(* Logix 5000 project; controller TEC_81 vendor 1 type 14 code 148 rev 36.11; software revision 36.00; part 4 of 4 *)
(* tags used below, declared in another part *)
   Safety_Close_Loop_ok : BOOL;
   TOF_STO_KinetixStorage1 : TIMER;
   Abrir_Prensa_CNC_1_Safety : BOOL;   // Abrir Prensa CNC 1
   Abrir_Prensa_CNC_2_Safety : BOOL;
   Cerrar_Prensa_CNC_1_Safety : BOOL;   // Cerrar Prensa CNC 1
   Cerrar_Prensa_CNC_2_Safety : BOOL;
   Close_Door_CNC_1_Safety : BOOL;   // Cerrar Puerta de CNC 1 Desde ArmorBlock
   Close_Door_CNC_2_Safety : BOOL;   // Cerrar Puerta de CNC 2 Desde ArmorBlock
   CycleStartDly : TIMER;
   EStops_OK : BOOL;
   Interlocks_Ok : BOOL;
   KUKA : TIMER;
   LigthCurtain_ok : BOOL;
   Paro_Emergencia_Almacen_1 : BOOL;   // Señal de paro para Torc Off Almacen 1
   Paro_Emergencia_Almacen_2 : BOOL;   // Señal de paro para Torc Off Almacen 2
   Pulse : TIMER;
   Reset_Almacen_1_Sfty : BOOL;
   Reset_Almacen_2_Sfty : BOOL;
   Reset_Principal_Sfty : BOOL;
   Reset_Salida_1_Sfty : BOOL;
   Safety_Test_Bit : DINT;
   SafetyReset_almacen_1 : BOOL;
   SafetyReset_almacen_2 : BOOL;
   SafetyReset_Principal : BOOL;
   SafetyReset_Salida_1 : BOOL;
   Storage_2 : BOOL;
   Storage_3 : BOOL;
   Storage_4 : BOOL;
   Storage_5 : BOOL;
   TOF_STO_KinetixStorage2 : TIMER;
   TT : BOOL;
(* SafetyProgram, continued *)

ROUTINE MainRoutine   (* ladder *)
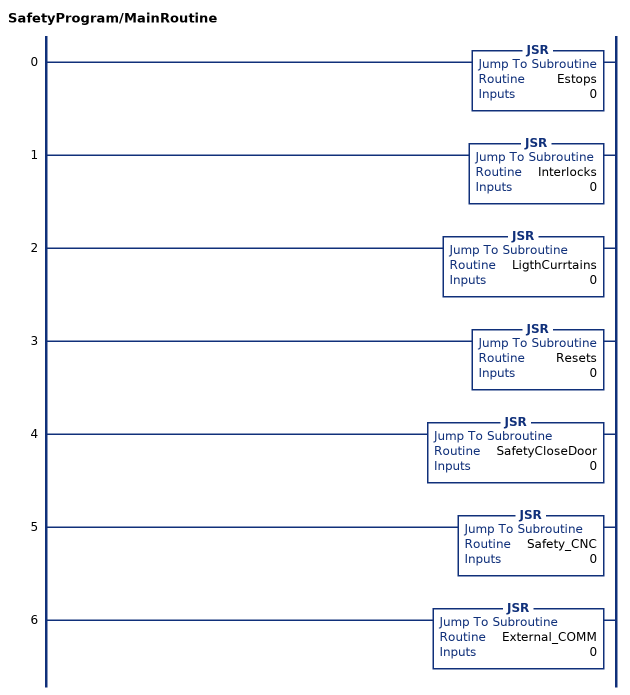
   0: JSR(Estops,0);
   1: JSR(Interlocks,0);
   2: JSR(LigthCurrtains,0);
   3: JSR(Resets,0);
   4: JSR(SafetyCloseDoor,0);
   5: JSR(Safety_CNC,0);
   6: JSR(External_COMM,0);
END_ROUTINE

ROUTINE Resets   (* ladder *)
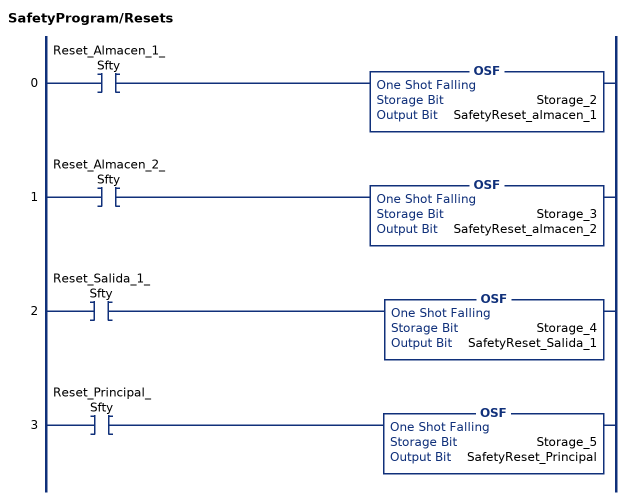
   0: XIC(Reset_Almacen_1_Sfty)OSF(Storage_2,SafetyReset_almacen_1);
   1: XIC(Reset_Almacen_2_Sfty)OSF(Storage_3,SafetyReset_almacen_2);
   2: XIC(Reset_Salida_1_Sfty)OSF(Storage_4,SafetyReset_Salida_1);
   3: XIC(Reset_Principal_Sfty)OSF(Storage_5,SafetyReset_Principal);
END_ROUTINE

ROUTINE Safety_CNC   (* ladder *)
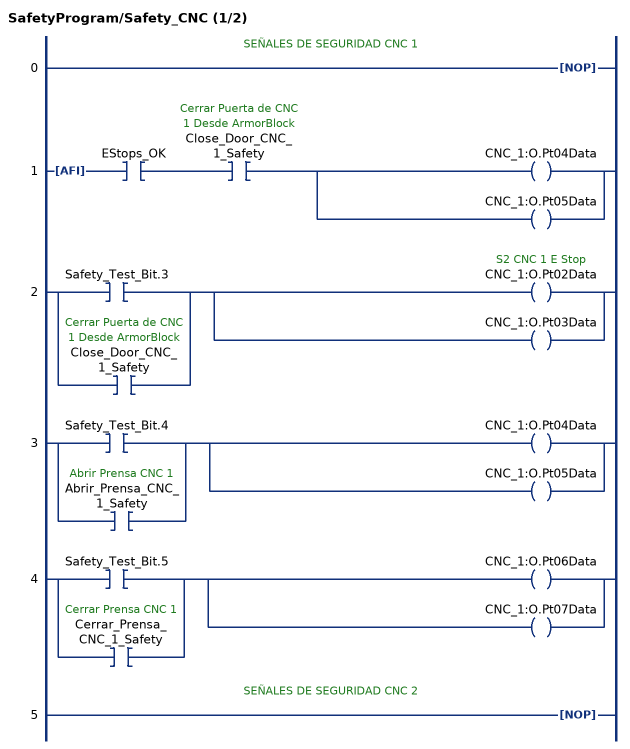
   // SEÑALES DE SEGURIDAD CNC 1
   0: NOP();
   1: AFI()XIC(EStops_OK)XIC(Close_Door_CNC_1_Safety)[OTE(CNC_1:O.Pt04Data) ,OTE(CNC_1:O.Pt05Data) ];
   2: [XIC(Safety_Test_Bit.3) ,XIC(Close_Door_CNC_1_Safety) ][OTE(CNC_1:O.Pt02Data) ,OTE(CNC_1:O.Pt03Data) ];
   3: [XIC(Safety_Test_Bit.4) ,XIC(Abrir_Prensa_CNC_1_Safety) ][OTE(CNC_1:O.Pt04Data) ,OTE(CNC_1:O.Pt05Data) ];
   4: [XIC(Safety_Test_Bit.5) ,XIC(Cerrar_Prensa_CNC_1_Safety) ][OTE(CNC_1:O.Pt06Data) ,OTE(CNC_1:O.Pt07Data) ];
   // SEÑALES DE SEGURIDAD CNC 2
   5: NOP();
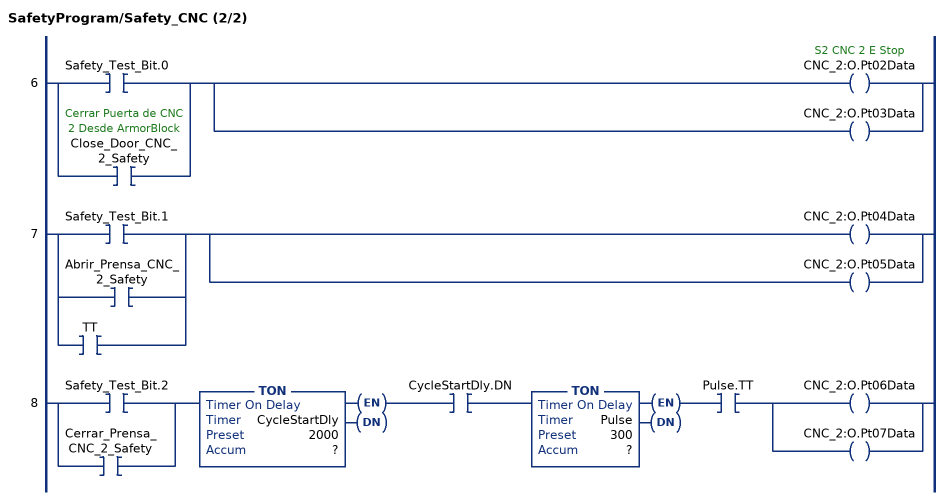
   6: [XIC(Safety_Test_Bit.0) ,XIC(Close_Door_CNC_2_Safety) ][OTE(CNC_2:O.Pt02Data) ,OTE(CNC_2:O.Pt03Data) ];
   7: [XIC(Safety_Test_Bit.1) ,XIC(Abrir_Prensa_CNC_2_Safety) ,XIC(TT) ][OTE(CNC_2:O.Pt04Data) ,OTE(CNC_2:O.Pt05Data) ];
   8: [XIC(Safety_Test_Bit.2) ,XIC(Cerrar_Prensa_CNC_2_Safety) ]TON(CycleStartDly,?,?)XIC(CycleStartDly.DN)TON(Pulse,?,?)XIC(Pulse.TT)[OTE(CNC_2:O.Pt06Data) ,OTE(CNC_2:O.Pt07Data) ];
END_ROUTINE

ROUTINE SafetyCloseDoor   (* ladder *)
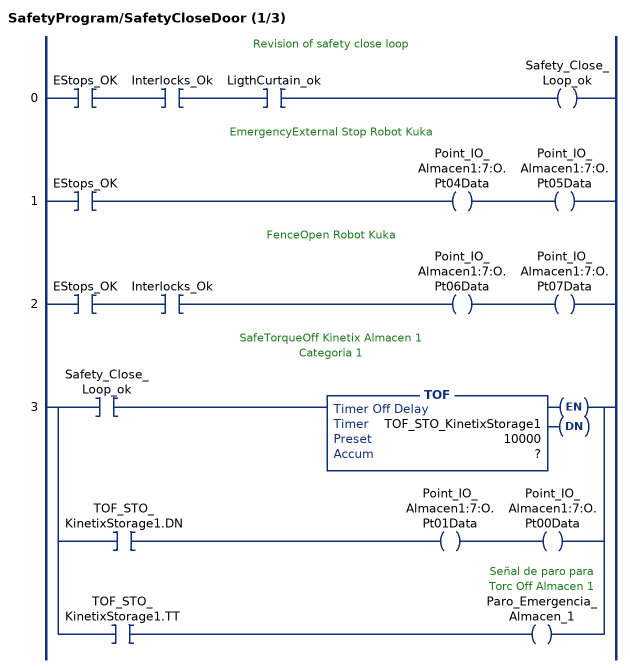
   // Revision of safety close loop
   0: XIC(EStops_OK)XIC(Interlocks_Ok)XIC(LigthCurtain_ok)OTE(Safety_Close_Loop_ok);
   // EmergencyExternal Stop Robot Kuka
   1: XIC(EStops_OK)OTE(Point_IO_Almacen1:7:O.Pt04Data)OTE(Point_IO_Almacen1:7:O.Pt05Data);
   // FenceOpen Robot Kuka
   2: XIC(EStops_OK)XIC(Interlocks_Ok)OTE(Point_IO_Almacen1:7:O.Pt06Data)OTE(Point_IO_Almacen1:7:O.Pt07Data);
   // SafeTorqueOff Kinetix Almacen 1
   // Categoria 1
   3: [XIC(Safety_Close_Loop_ok) TOF(TOF_STO_KinetixStorage1,?,?) ,XIC(TOF_STO_KinetixStorage1.DN) OTE(Point_IO_Almacen1:7:O.Pt01Data) OTE(Point_IO_Almacen1:7:O.Pt00Data) ,XIC(TOF_STO_KinetixStorage1.TT) OTE(Paro_Emergencia_Almacen_1) ];
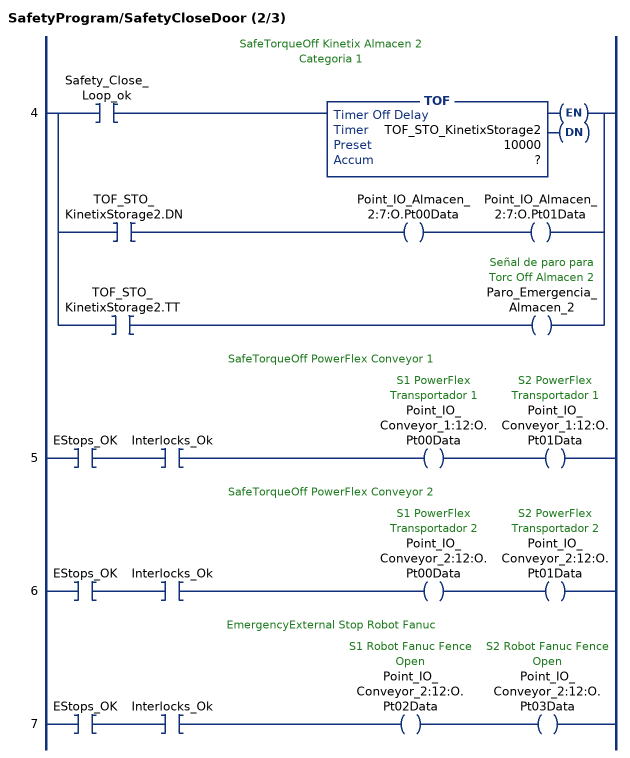
   // SafeTorqueOff Kinetix Almacen 2
   // Categoria 1
   4: [XIC(Safety_Close_Loop_ok) TOF(TOF_STO_KinetixStorage2,?,?) ,XIC(TOF_STO_KinetixStorage2.DN) OTE(Point_IO_Almacen_2:7:O.Pt00Data) OTE(Point_IO_Almacen_2:7:O.Pt01Data) ,XIC(TOF_STO_KinetixStorage2.TT) OTE(Paro_Emergencia_Almacen_2) ];
   // SafeTorqueOff PowerFlex Conveyor 1
   5: XIC(EStops_OK)XIC(Interlocks_Ok)OTE(Point_IO_Conveyor_1:12:O.Pt00Data)OTE(Point_IO_Conveyor_1:12:O.Pt01Data);
   // SafeTorqueOff PowerFlex Conveyor 2
   6: XIC(EStops_OK)XIC(Interlocks_Ok)OTE(Point_IO_Conveyor_2:12:O.Pt00Data)OTE(Point_IO_Conveyor_2:12:O.Pt01Data);
   // EmergencyExternal Stop Robot Fanuc
   7: XIC(EStops_OK)XIC(Interlocks_Ok)OTE(Point_IO_Conveyor_2:12:O.Pt02Data)OTE(Point_IO_Conveyor_2:12:O.Pt03Data);
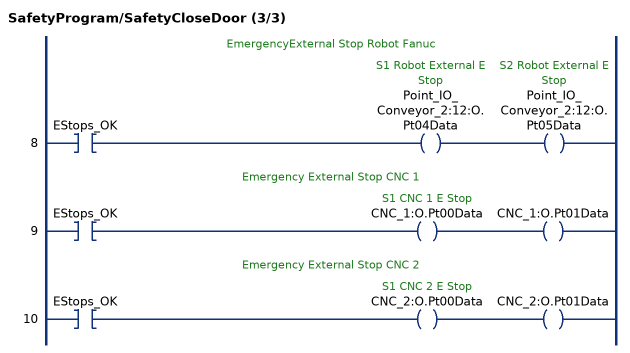
   // EmergencyExternal Stop Robot Fanuc
   8: XIC(EStops_OK)OTE(Point_IO_Conveyor_2:12:O.Pt04Data)OTE(Point_IO_Conveyor_2:12:O.Pt05Data);
   // Emergency External Stop CNC 1
   9: XIC(EStops_OK)OTE(CNC_1:O.Pt00Data)OTE(CNC_1:O.Pt01Data);
   // Emergency External Stop CNC 2
   10: XIC(EStops_OK)OTE(CNC_2:O.Pt00Data)OTE(CNC_2:O.Pt01Data);
END_ROUTINE
END_PROGRAM
